// TIA Portal V18 export
// export: Created 2026-06-07T17:03:10.303355Z, ExportSetting WithDefaults, DisplayName Totally Integrated Automation Portal, DisplayVersion V18, DisplayName TIA Portal Openness, DisplayVersion V18, DisplayName TIA Portal Version Control Interface, DisplayVersion V18, DisplayName STEP 7 Professional, DisplayVersion V18, DisplayName STEP 7 Safety, DisplayVersion V18, DisplayName WinCC Professional, DisplayVersion V18
DATA_BLOCK "DB_MB_Client_Data"   // DB10
TITLE = DB_MB_Client_Data
{ S7_Optimized_Access := 'FALSE' }
VERSION : 0.1
// DB communication via Modbus TCP
// stored: AutoNumber false, IsOnlyStoredInLoadMemory false, IsWriteProtectedInAS false
   VAR
      Send_Words : Array[0..2] of Int;
      Recv_Words : Array[0..9] of Int;
   END_VAR
BEGIN
END_DATA_BLOCK
